// TwinCAT 3 PLC project HeaterDemo
// ProgramVersion: 3.1.0.9
// libraries:
//   Tc2_ControllerToolbox,newest,Beckhoff Automation GmbH
//   Tc2_Standard,newest,Beckhoff Automation GmbH
//   Tc2_System,newest,Beckhoff Automation GmbH
//   Tc2_TempController,newest,Beckhoff Automation GmbH
//   Tc2_Utilities,newest,Beckhoff Automation GmbH
//   Tc3_Module,newest,Beckhoff Automation GmbH
//   VisuDialogs, * (System)
// project tree:
//   Data types/ E_TunePreSets.TcDUT, ST_TuneParams.TcDUT
//   / GlobalImagePool.TcIPO (not stored), GlobalTextList.TcGTLO, Standard.TcTTO, Visualization Manager.TcVMO (not stored)
//   POUs/ MAIN.TcPOU
//   Visualizations/ HMI.TcVIS
// real-time tasks:
//   TASK Standard: cycle T#10ms, priority 20, ADS port 350

CONFIGURATION HeaterDemo
    RESOURCE PLC ON TwinCAT3
        TASK Standard(INTERVAL := T#10ms, PRIORITY := 20);
        PROGRAM MAIN WITH Standard : MAIN;
    END_RESOURCE
END_CONFIGURATION

// ---- Data types/E_TunePreSets.TcDUT
{attribute 'qualified_only'}
{attribute 'strict'}
TYPE E_TunePreSets :
(
	Fast := 0, 	// Fast settling with overshoots of 10%-20%
	Slow,		// Slower settling with low overshoot
	Asymptotic	//Almost asymptotic settling with extremely small overshoot
);
END_TYPE

// ---- Data types/ST_TuneParams.TcDUT
TYPE ST_TuneParams :
STRUCT
	fKp			:LREAL;
	fTn			:LREAL;
	fTv			:LREAL;
	fTd			:LREAL;
END_STRUCT
END_TYPE

// ---- POUs/MAIN.TcPOU
PROGRAM MAIN
VAR
	// Safety / Estop override
	bEnabled: BOOL;							// manually turn off / disable output 

	// Temp control FB vars
	fbTempContrl: FB_CTRL_TempController;	
	nControllerMode: E_CTRL_MODE;			// := eCTRL_MODE_TUNE; (* start with tuning *)
	bHeaterOn: BOOL;						// PWM digital output
	rTempF: REAL;							// Actual temperature feedback
	
	fSetPoint: REAL :=100.0;				// if using tuning, setpoint must be > .8 of (initial + tuning step)
	bHeat: BOOL;							// output of controller 

	// simulation model vars
	rTempBuf: ARRAY[1..iMaxDelay] OF REAL; 	// array for delay
	iDelay: UINT:=500;						// thermal temp delay --> 500 is 5 sec
	rHeatGain: REAL := 0.05;				// how big is heater
	rCoolOffGain: REAL := 0.0001;			// ambient cooling effect
	bResetModel: BOOL;						// reset model to zero
	
	// tuning PID gains
	sParaControlExternal	: ST_CTRL_ParaController := (
		// for use when NOT starting with tuning -- values need
		// to be calc'd or determined once with autotuning Controller parameter set - heating 
		KpHeat			:= 32.36,
		TnHeat			:= T#51S502MS,
		TvHeat			:= T#10S815MS,
		TdHeat			:= T#2S704MS,

		// Controller parameter set - cooling - not used in this example
		KpCool			:= 0,
		TnCool			:= T#0S,
		TvCool			:= T#0S,
		TdCool			:= T#0S
		);


	// controller parameter struct (populated)
	stCntrlParam	: ST_CTRL_TempCtrlParameter := (		
		
		(* general parameters 													 *)
		iMode					:= 1,											(* 1=heating, 2=cooling, 3=heating&cooling *)
		iReactionOnFailure		:= eCTRL_ReactionOnFailure_StopController,		(* 0=controller off, 1=manual op, 2=yMin, 3=yMax *)
	
		bSelCtrlParameterSet	:= FALSE,										(* FALSE = internal set, TRUE = external set *)
	
		dwAlarmSupp				:= 16#0000EFFF,									(* alarm suppression *)
		tCtrlCycleTime			:= T#500MS,										(* controller cycle time *)
		tTaskCycleTime			:= T#10MS,										(* plc task cycle time *)
		
		(* tuning parameters 													 *)
		iTuningMode				:= 1,											(* only heating, only cooling, first heating then cooling or vice versa *)
	
		tTuneStabilisation		:= T#20S,										(* wait for a stable system *)
	
		fEndTunePercentHeating	:= 80.0,										(* switch to closed loop control when X > 0.8*W *)
		fYTuneHeating			:= 100.0,										(* step change while tuning operation *)
		fYStableHeating			:= 0.0,											(* tuning operation *)
	
		fEndTunePercentCooling	:= 20.0,										(* switch to closed loop control when X < 0.2*W *)
		fYTuneCooling			:= 0.0,											(* step change while tuning operation *)
		fYStableCooling			:= 0.0,											(* tuning operation *)
		fScalingFactor			:= 1.0,											(* Scaling factor for KP heating/cooling *)
		
		(* setpoint parameters 													 *)
		fWMin					:= 0.0,											(* lower limit *)
		fWMax					:= 300.0,										(* upper limit *)
	
		(* start up *)
		bEnableSoftStart		:= FALSE,										(* FALSE = no soft start, TRUE = soft start *)
		bEnableRamping			:= FALSE,										(* FALSE = no ramping, TRUE = ramping *)
	
		fWStartUp				:= 0.0,											(* soft start plateau setpoint *)
		tStartUp				:= T#0MS,										(* soft start waiting time*)
		bStartUpRamping			:= FALSE,										(* enable ramping while start up phase *)
		fWStartUpVeloPos		:= 1.0,											(* max gradient for increasing setpoint in start up phase*)
		fWStartUpVeloNeg		:= 1.0,											(* max gradient for decreasing setpoint in start up phase *)
	
		fWVeloPos				:= 1.0,											(* max gradient for increasing setpoint *)
		fWVeloNeg				:= 1.0,											(* max gradient for decreasing setpoint *)	
	
		(* actual value parameters     											 *)
		bFilter 				:= FALSE,
		tFilter					:= T#0S,
		
		(* deadband parameters     												 *)
		bDeadband				:= FALSE,
		fEDeadband				:= 0.0,											(* deadband *)
		
		(* control value parameters     										 *)
		fYMin					:= 0.0,											(* lower limit *)
		fYMax					:= 100.0,										(* upper limit *)
		fYManual				:= 0.0,									 		(* manual operation*)
		fYOnFailure				:= 0.0,											(* control value on failure *)
	
		tPWMCycleTime			:= t#1s,										(* PWM: period *)
		tPWMMinOffTime			:= t#0s,										(* PWM: min off time *)
		tPWMMinOnTime			:= t#0s,										(* PWM: min on time *)
		tPWMWaitingTime			:= t#0s,										(* PWM: min waiting time *) (* not yet implemented !!!!*)
	
		fYThresholdOff			:= 0.0,											(* 3-Point: Off threshold *)
		fYThresholdOn			:= 0.0,											(* 3-Point: On threshold *)
	
		nCyclesForSwitchOver	:= 100,
	
		(* controller settings			     									 *)
		bEnablePreController 	:= FALSE,										(* enable precontroller *)
		bEnableZones 			:= FALSE,										(* enable zone around setpoint with open loop control *)
		bEnableCVFilter 		:= FALSE,										(* enable filter for CV (type see iFilterType) *)
		iFilterType 			:= eCTRL_FilterType_FIRSTORDER,			 		(* filtertype of CV filter *)
		iControllerType 		:= eCTRL_ControllerType_PID,					(* used controller normally PID *)
		
		
		(* min max temperatures	     											 *)
		TempLow					:= -5.0,
		TempLowLow				:= -10.0,
		TempHigh				:= 5.0,
		TempHighHigh			:= 10.0,
		TempAbsoluteHigh		:= 300.0,
		TempAbsoluteLow			:= 0.0,	
		
		(* internal tuning parameters *)
		fTuneKp					:= 1.2,
		fTuneTn					:= 2.0,
		fTuneTv					:= 0.42,
		fTuneTd					:= 0.25
		);
		
	bLoadTuneParamSet			:BOOL;
	SelectedParamSetToLoad		:E_TunePreSets;	
END_VAR
VAR CONSTANT
	TuneParamPreSets: ARRAY [E_TunePreSets.Fast..E_TunePreSets.Asymptotic] OF ST_TuneParams := 
	[	(fKp := 1.2, fTn := 2.0, fTv := 0.42, fTd := 0.25), 
		(fKp := 1.0, fTn := 2.5, fTv := 0.42, fTd := 0.25), 
		(fKp := 0.5, fTn := 3.0, fTv := 1.0, fTd := 0.25)
	];	
	iMaxDelay		:UINT := 6000;	// 6000 is 60 seconds
END_VAR


TempControl();

(* manually disable heater output if needed *)
IF bEnabled AND bHeat THEN
	bHeaterOn := TRUE;
ELSE
	bHeaterOn := FALSE;
END_IF

IF bLoadTuneParamSet THEN
	bLoadTuneParamSet	:=FALSE;
	stCntrlParam.fTuneKp:=TuneParamPreSets[SelectedParamSetToLoad].fKp;
	stCntrlParam.fTuneTd:=TuneParamPreSets[SelectedParamSetToLoad].fTd;
	stCntrlParam.fTuneTn:=TuneParamPreSets[SelectedParamSetToLoad].fTn;
	stCntrlParam.fTuneTv:=TuneParamPreSets[SelectedParamSetToLoad].fTv;
	
END_IF

// simulated process with thermal time delay
rTempBuf[1] := rTempBuf[1] + BOOL_TO_REAL(bHeaterOn)* rHeatGain - (rTempBuf[1]*rCoolOffGain);
rTempF := rTempBuf[iDelay];
MEMCPY(destAddr:= ADR(rTempBuf[2]), srcAddr:= ADR(rTempBuf[1]), n:= (iMaxDelay-1)*SIZEOF(rTempBuf[1]));

IF bResetModel THEN
	bResetModel:=FALSE;
	MEMSET(destAddr:= ADR(rTempBuf[1]), fillByte:= 16#00, n:= (iMaxDelay)*SIZEOF(rTempBuf[1]));
END_IF

ACTION TempControl:
fbTempContrl(
    eCtrlMode := nControllerMode,
    fW1 := fSetPoint,
    fX := rTempF,
    sParaControllerExternal := sParaControlExternal,
    sControllerParameter := stCntrlParam); // FB_CTRL_TempController
bHeat := fbTempContrl.bYPWMPos;
END_ACTION

END_PROGRAM

// ---- GlobalTextList.TcGTLO
TEXTLIST GlobalTextList
  222 = '%1.2f'
  941 = '%1.5f'
  232 = '%1.6f'
  230 = '%s'
  229 = 'Active'
  224 = 'Actual Temp'
  427 = 'Ambient cool off effect'
  316 = 'bEnable'
  221 = 'bRun'
  223 = 'Controller FB error'
  919 = 'fTuneKp =  %1.4f'
  220 = 'fTuneTd =  %s'
  24 = 'fTuneTd=  %s'
  614 = 'fTuneTn =  %s'
  203 = 'fTuneTv =  %s'
  617 = 'Heater Power'
  227 = 'Idle'
  733 = 'Internal gains (from tuning)'
  708 = 'internal tuning parameters'
  643 = 'KpHeat =  %1.4f'
  657 = 'KpHeat =  %s'
  676 = 'Reset'
  554 = 'Reset Act Temp = 0'
  225 = 'SetPoint Temp'
  239 = 'Simulation model'
  515 = 'TdHeat =  %s'
  742 = 'Thermal delay (500 = 5 sec)'
  936 = 'TnHeat =  %s'
  228 = 'Tune'
  226 = 'Tuned'
  244 = 'TvHeat =  %s'
  231 = 'Use Ext Params'
END_TEXTLIST

// ---- Visualizations/HMI.TcVIS
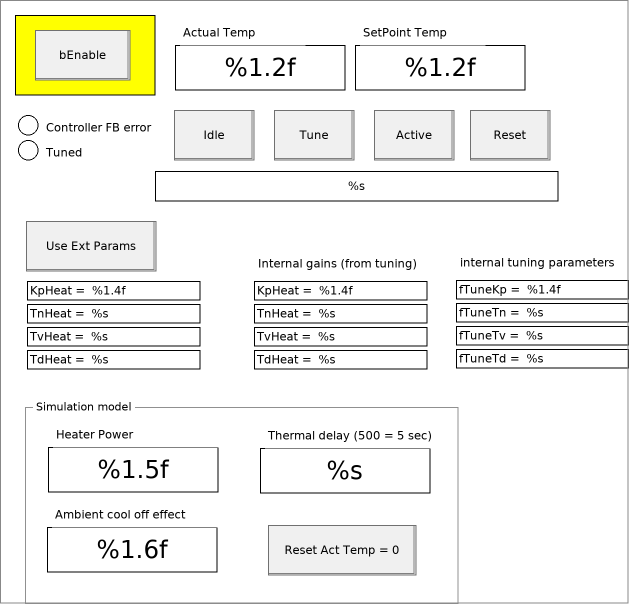
VISUALIZATION HMI  // 629x604
    Rectangle (15,15 140x80), colour toggle: MAIN.bEnabled
    Button (35,30 95x50), "bEnable", pressed state: MAIN.bEnabled
        toggle MAIN.bEnabled
    Rectangle (175,45 170x45), "%1.2f", text variable: MAIN.rTempF, colour toggle: MAIN.bHeaterOn
    Ellipse (18,115 20x20), colour toggle: (MAIN.fbTempContrl.bError) <> 0
    Rectangle (43,115 114x25), "Controller FB error"
    Rectangle (180,20 125x25), "Actual Temp"
    Rectangle (355,45 170x45), "%1.2f", text variable: MAIN.fSetPoint
        OnMouseDown: write the text variable via VisuDialogs.Numpad
    Rectangle (360,20 125x25), "SetPoint Temp"
    Ellipse (18,140 20x20), colour toggle: (MAIN.fbTempContrl.bTuned) <> 0
    Rectangle (43,140 69x25), "Tuned"
    Button (174,110 80x50), "Idle"
        OnMouseUp: execute { MAIN.nControllerMode:=E_CTRL_MODE.eCTRL_MODE_IDLE; }
    Button (274,110 80x50), "Tune"
        OnMouseUp: execute { MAIN.nControllerMode:=E_CTRL_MODE.eCTRL_MODE_TUNE; }
    Button (374,110 80x50), "Active"
        OnMouseUp: execute { MAIN.nControllerMode:=E_CTRL_MODE.eCTRL_MODE_ACTIVE; }
    Rectangle (155,171 403x30), "%s", text variable: MAIN.fbTempContrl.eCtrlState
    Button (26,221 130x50), "Use Ext Params", pressed state: MAIN.stCntrlParam.bSelCtrlParameterSet
        toggle MAIN.stCntrlParam.bSelCtrlParameterSet
    Button (470,110 80x50), "Reset"
        OnMouseUp: execute { MAIN.nControllerMode:=E_CTRL_MODE.eCTRL_MODE_RESET; }
    Rectangle (27,281 173x19), "KpHeat = %1.4f", text variable: MAIN.sParaControlExternal.KpHeat
        OnMouseDown: write the text variable via Edit
    Rectangle (27,304 173x19), "TnHeat = %s", text variable: MAIN.sParaControlExternal.TnHeat
        OnMouseDown: write the text variable via Edit
    Rectangle (27,327 173x19), "TvHeat = %s", text variable: MAIN.sParaControlExternal.TvHeat
        OnMouseDown: write the text variable via Edit
    Rectangle (27,350 173x19), "TdHeat = %s", text variable: MAIN.sParaControlExternal.TdHeat
        OnMouseDown: write the text variable via Edit
    Rectangle (254,281 173x19), "KpHeat = %1.4f", text variable: MAIN.fbTempContrl.sParaControllerInternal.KpHeat
        OnMouseDown: write the text variable via Edit
    Rectangle (254,304 173x19), "TnHeat = %s", text variable: MAIN.fbTempContrl.sParaControllerInternal.TnHeat
        OnMouseDown: write the text variable via Edit
    Rectangle (254,327 173x19), "TvHeat = %s", text variable: MAIN.fbTempContrl.sParaControllerInternal.TvHeat
        OnMouseDown: write the text variable via Edit
    Rectangle (254,350 173x19), "TdHeat = %s", text variable: MAIN.fbTempContrl.sParaControllerInternal.TdHeat
        OnMouseDown: write the text variable via Edit
    Rectangle (255,251 167x25), "Internal gains (from tuning)"
    GroupBox (25,399 433x205), "Simulation model"
        Rectangle (23,48 170x45), "%1.5f", text variable: MAIN.rHeatGain
            OnMouseDown: write the text variable via InputWithLimits, min 0.00001, max 2
        Rectangle (28,23 180x25), "Heater Power"
        Rectangle (235,49 170x45), "%s", text variable: MAIN.iDelay
            OnMouseDown: write the text variable via InputWithLimits, min 1, max 6000
        Rectangle (22,128 170x45), "%1.6f", text variable: MAIN.rCoolOffGain
            OnMouseDown: write the text variable via InputWithLimits, min 0.000001, max 1
        Button (243,126 148x50), "Reset Act Temp = 0", pressed state: MAIN.stCntrlParam.bSelCtrlParameterSet
            toggle MAIN.bResetModel
    Rectangle (265,423 180x25), "Thermal delay (500 = 5 sec)"
    Rectangle (52,502 180x25), "Ambient cool off effect"
    Rectangle (456,280 173x19), "fTuneKp = %1.4f", text variable: MAIN.stCntrlParam.fTuneKp
        OnMouseDown: write the text variable via Edit
    Rectangle (456,303 173x19), "fTuneTn = %s", text variable: MAIN.stCntrlParam.fTuneTn
        OnMouseDown: write the text variable via Edit
    Rectangle (456,326 173x19), "fTuneTv = %s", text variable: MAIN.stCntrlParam.fTuneTv
        OnMouseDown: write the text variable via Edit
    Rectangle (456,349 173x19), "fTuneTd = %s", text variable: MAIN.stCntrlParam.fTuneTd
        OnMouseDown: write the text variable via Edit
    Rectangle (457,250 167x25), "internal tuning parameters"
END_VISUALIZATION
